FUNCTION_BLOCK FB_VFD
VAR_INPUT
END_VAR
VAR_OUTPUT
END_VAR
VAR
END_VAR

END_FUNCTION_BLOCK

(* stored: Version 1.1.0.1, ProductVersion 3.1.4024.12
   POU FB_VFD: Id {3dc147eb-3dde-4052-8db8-ee0200a73c1f}, SpecialFunc None *)
